// TIA Portal V20 export
DATA_BLOCK "SBK10"   // DB328
// stored: MemoryReserve 100
   VAR
      "SAFETY DOOR LOCK7.INPUT" : Bool := TRUE;
      SPARE_5 : Bool := TRUE;
      "SAFETY DOOR LOCK9.INPUT" : Bool := TRUE;
      SPARE : Bool := FALSE;
      "SAFETY DOOR LOCK7.INPUT_1" : Bool := FALSE;
      SPARE_1 : Bool := FALSE;
      "SAFETY DOOR LOCK9.INPUT_1" : Bool := FALSE;
      SPARE_2 : Bool := FALSE;
      "SAFETY DOOR LOCK7.OUTPUT" : Bool := FALSE;
      SPARE_3 : Bool := FALSE;
      "SAFETY DOOR LOCK9.OUTPUT" : Bool := FALSE;
   END_VAR
BEGIN
END_DATA_BLOCK
